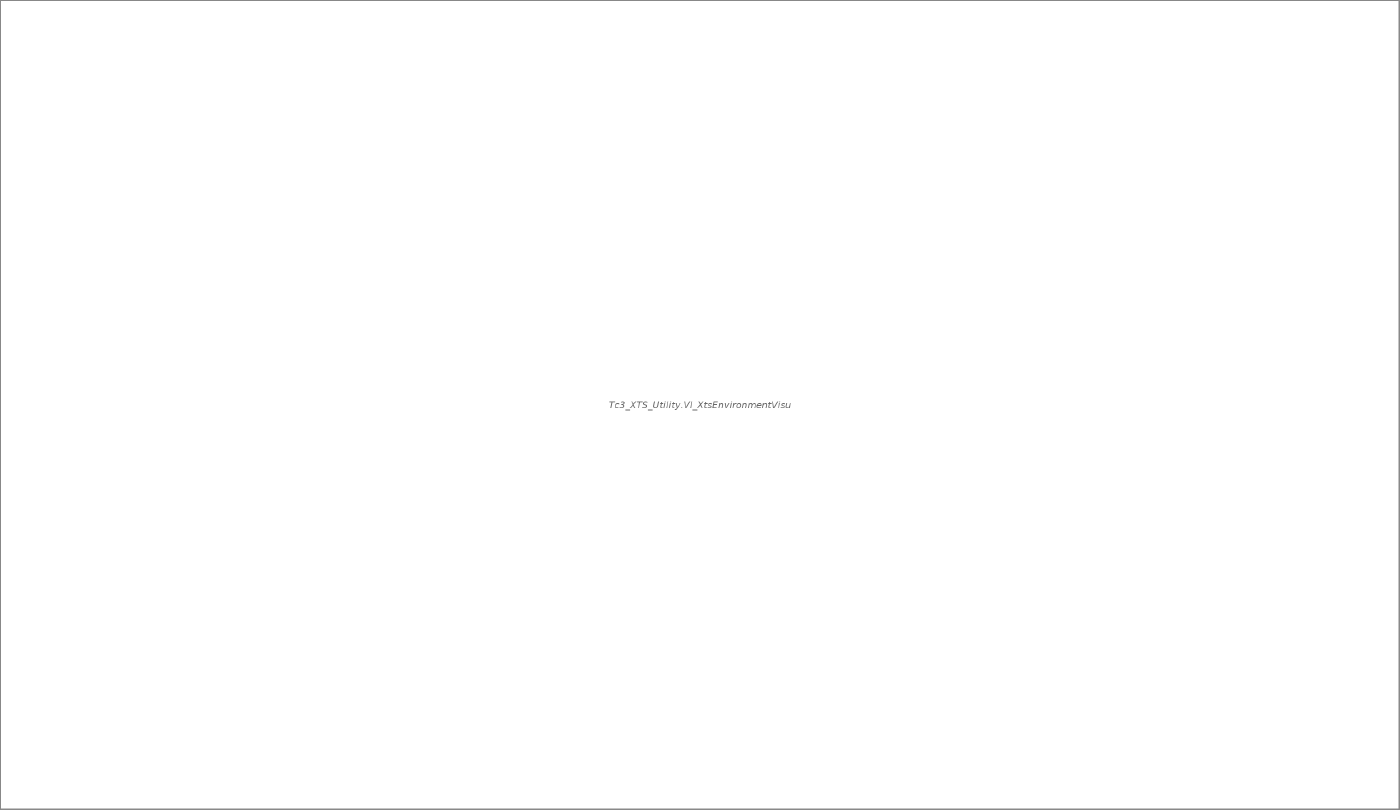
VISUALIZATION PageXtsEnviroment  // 1520x880
    Frame (0,0 1520x880)
        shows Tc3_XTS_Utility.VI_XtsEnvironmentVisu()
END_VISUALIZATION

(* stored: Version 1.1.0.1, ProductVersion 3.1.4024.9
   Visu PageXtsEnviroment: Id {1a00a279-29c5-4a91-9d7b-c0052a152729} *)
